// TIA Portal V15.1 export
// export: Created 2024-05-17T05:38:36.150876Z, ExportSetting WithDefaults, DisplayName Totally Integrated Automation Portal, DisplayVersion V15.1 Update 5, DisplayName TIA Portal Openness, DisplayVersion V15.1 Update 5, DisplayName SINAMICS Startdrive Advanced, DisplayVersion V15.1, DisplayName G130, G150, S120, S150, SINAMICS MV, S210, DisplayVersion V15.1, DisplayName G110M, G120, G120C, G120D, G120P, DisplayVersion V15.1, DisplayName STEP 7 Professional, DisplayVersion V15.1 Update 5, DisplayName STEP 7 Safety, DisplayVersion V15.1, DisplayName WinCC Professional, DisplayVersion V15.1 Update 5, DisplayName SIMATIC Visualization Architect, DisplayVersion V15.1
FUNCTION_BLOCK "LProcGeneralFunc"   // FB1738, FBD
TITLE = LProcGeneralFunc
{ S7_Optimized_Access := 'TRUE' }
AUTHOR : VCC
FAMILY : Control
NAME : Genfunc
VERSION : 0.1
// ================================================================================
// This module handles General Reverse Switch, General High Speed and Lamptest.
// It will also give the user and 8 bit interface for project specific functions.
// ================================================================================
// stored: AutoNumber false, IsIECCheckEnabled false, IsRetainMemResEnabled false, MemoryReserve 100, SetENOAutomatically False, UDAEnableTagReadback false
   VAR_INPUT
      I_GenRevSw { ExternalAccessible := 'False'; ExternalVisible := 'False'; ExternalWritable := 'False'} : Bool;   // General reverse switch
      I_GenHighSpeed { ExternalAccessible := 'False'; ExternalVisible := 'False'; ExternalWritable := 'False'} : Bool;   // General high speed
      I_Lamptest { ExternalAccessible := 'False'; ExternalVisible := 'False'; ExternalWritable := 'False'} : Bool;   // Lamptest PB
      I_ManualMode { ExternalAccessible := 'False'; ExternalVisible := 'False'; ExternalWritable := 'False'} : Bool := TRUE;   // Manual mode active
      I_LamptestSec { ExternalAccessible := 'False'; ExternalVisible := 'False'; ExternalWritable := 'False'} : Int := 60;   // The number of seconds that Lamptest will be on (Sec)
   END_VAR
   VAR_OUTPUT
      O_GeneralFunc : Word;   // General functions
      O_Lamptest { ExternalAccessible := 'False'; ExternalVisible := 'False'; ExternalWritable := 'False'} : Bool;   // Lamptest
      O_LamptestSteady { ExternalAccessible := 'False'; ExternalVisible := 'False'; ExternalWritable := 'False'} : Bool;   // Lamptest always on
      O_GenHighSpeed { ExternalAccessible := 'False'; ExternalVisible := 'False'; ExternalWritable := 'False'} : Bool;   // General High Speed
      O_GenRevSwitch { ExternalAccessible := 'False'; ExternalVisible := 'False'; ExternalWritable := 'False'} : Bool;   // Reverse Switch
      O_GenReverseAlarm { ExternalAccessible := 'False'; ExternalVisible := 'False'; ExternalWritable := 'False'} : Bool;   // Alarm when general reverse switch is ON while NOT in Manual mode
   END_VAR
   VAR DB_SPECIFIC
      H_HMIGenFuncCmd : Word;   // General function commands from HMI
      AutoMode { ExternalAccessible := 'False'; ExternalVisible := 'False'; ExternalWritable := 'False'} : Bool;   // Auto mode
      AutoSel { ExternalAccessible := 'False'; ExternalVisible := 'False'; ExternalWritable := 'False'} : Bool;   // Auto is selected
      AlarmAB { ExternalAccessible := 'False'; ExternalVisible := 'False'; ExternalWritable := 'False'} : Bool;   // Alarm A or B is active
      HMIGenHighSpeed { ExternalAccessible := 'False'; ExternalVisible := 'False'; ExternalWritable := 'False'} : Bool;   // General High Speed for manual movement
      HMILamptest { ExternalAccessible := 'False'; ExternalVisible := 'False'; ExternalWritable := 'False'} : Bool;   // Lamptest
      GenHighSpeedSelected { ExternalAccessible := 'False'; ExternalVisible := 'False'; ExternalWritable := 'False'} : Bool;   // General high speed is selected
      LamptestSelected : Bool;   // Lamptest is selected
      PulseLamptest { ExternalAccessible := 'False'; ExternalVisible := 'False'; ExternalWritable := 'False'} : Bool;   // Pulse for lamptest
      PulseGenHighSpeed { ExternalAccessible := 'False'; ExternalVisible := 'False'; ExternalWritable := 'False'} : Bool;   // Pulse General high speed
      TimerLamptest { ExternalAccessible := 'False'; ExternalVisible := 'False'; ExternalWritable := 'False'} : Bool;   // Timer for Lamptest
      LamptestSec { ExternalAccessible := 'False'; ExternalVisible := 'False'; ExternalWritable := 'False'} : DInt;   // Lamptest on for xxx milliesec
      LamptestMillieSec { ExternalAccessible := 'False'; ExternalVisible := 'False'; ExternalWritable := 'False'} : DInt;   // Converted value
   END_VAR
   VAR
      TimerLampTestSel { ExternalAccessible := 'False'; ExternalVisible := 'False'; ExternalWritable := 'False'; S7_SetPoint := 'True'} : "LTimer";
   END_VAR
   VAR_TEMP
      SetLamptest : Bool;   // Set Lamptest
      ResetLamptest : Bool;   // Reset Lamptest
      ElapseTime : DInt;   // Elapse time for Lamptest
   END_VAR
   VAR_TEMP   // added for the SCL form of the ladder/FBD networks
      _w1 : Bool;
      _w2 : Bool;
   END_VAR
BEGIN

REGION Network 1: **** 1 - Inputs **** Extract the general functions from HMI
   // Extract the general functions from HMI
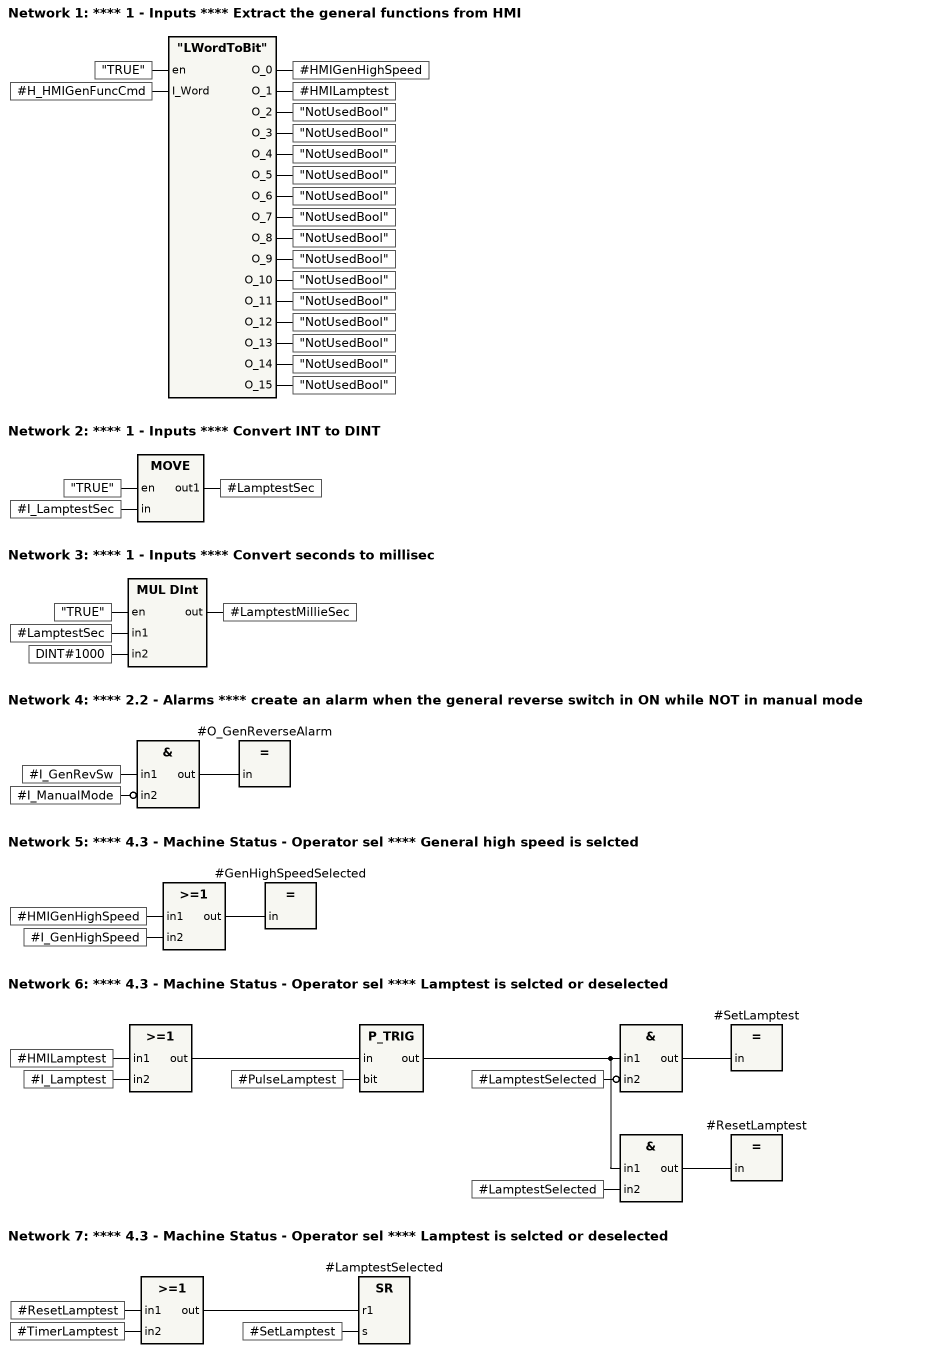
   IF "TRUE" THEN
       "LWordToBit"(I_Word := #H_HMIGenFuncCmd,
                    O_0 => #HMIGenHighSpeed,
                    O_1 => #HMILamptest,
                    O_2 => "NotUsedBool",
                    O_3 => "NotUsedBool",
                    O_4 => "NotUsedBool",
                    O_5 => "NotUsedBool",
                    O_6 => "NotUsedBool",
                    O_7 => "NotUsedBool",
                    O_8 => "NotUsedBool",
                    O_9 => "NotUsedBool",
                    O_10 => "NotUsedBool",
                    O_11 => "NotUsedBool",
                    O_12 => "NotUsedBool",
                    O_13 => "NotUsedBool",
                    O_14 => "NotUsedBool",
                    O_15 => "NotUsedBool");
   END_IF;
END_REGION

REGION Network 2: **** 1 - Inputs **** Convert INT to DINT
   // Convert INT to DINT
   IF "TRUE" THEN #LamptestSec := #I_LamptestSec; END_IF;
END_REGION

REGION Network 3: **** 1 - Inputs **** Convert seconds to millisec
   // Convert seconds to millisec
   IF "TRUE" THEN #LamptestMillieSec := #LamptestSec * DINT#1000; END_IF;
END_REGION

REGION Network 4: **** 2.2 - Alarms **** create an alarm when the general reverse switch in ON while NOT in manual mode
   // create an alarm when the general reverse switch in ON while NOT in manual mode
   #O_GenReverseAlarm := #I_GenRevSw AND NOT #I_ManualMode;
END_REGION

REGION Network 5: **** 4.3 - Machine Status - Operator sel **** General high speed is selcted
   // General high speed is selcted
   #GenHighSpeedSelected := #HMIGenHighSpeed OR #I_GenHighSpeed;
END_REGION

REGION Network 6: **** 4.3 - Machine Status - Operator sel **** Lamptest is selcted or deselected
   // Lamptest is selcted or deselected
   #_w1 := #HMILamptest OR #I_Lamptest;
   #_w2 := #_w1 AND NOT #PulseLamptest;   // rising edge
   #PulseLamptest := #_w1;
   #SetLamptest := #_w2 AND NOT #LamptestSelected;
   #ResetLamptest := #_w2 AND #LamptestSelected;
END_REGION

REGION Network 7: **** 4.3 - Machine Status - Operator sel **** Lamptest is selcted or deselected
   // Lamptest is selcted or deselected
   IF #SetLamptest THEN
       #LamptestSelected := TRUE;   // SR flip-flop
   END_IF;
   IF #ResetLamptest OR #TimerLamptest THEN #LamptestSelected := FALSE; END_IF;
END_REGION

REGION Network 8: **** 4.3 - Machine Status - Operator sel **** Timer for Lamptest
   // Timer for Lamptest
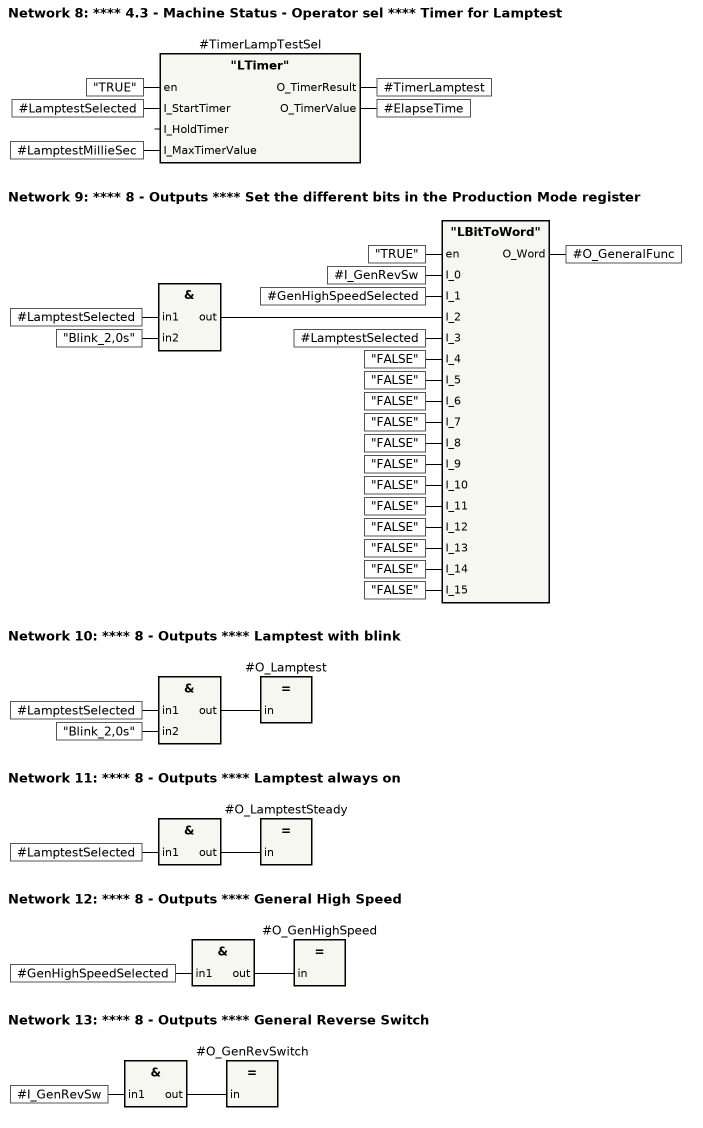
   IF "TRUE" THEN
       #TimerLampTestSel(I_StartTimer := #LamptestSelected,   // "LTimer"
                         I_MaxTimerValue := #LamptestMillieSec,
                         O_TimerResult => #TimerLamptest,
                         O_TimerValue => #ElapseTime);
   END_IF;
END_REGION

REGION Network 9: **** 8 - Outputs **** Set the different bits in the Production Mode register
   // Set the different bits in the Production Mode register
   IF "TRUE" THEN
       "LBitToWord"(I_0 := #I_GenRevSw,
                    I_1 := #GenHighSpeedSelected,
                    I_2 := #LamptestSelected AND "Blink_2,0s",
                    I_3 := #LamptestSelected,
                    I_4 := "FALSE",
                    I_5 := "FALSE",
                    I_6 := "FALSE",
                    I_7 := "FALSE",
                    I_8 := "FALSE",
                    I_9 := "FALSE",
                    I_10 := "FALSE",
                    I_11 := "FALSE",
                    I_12 := "FALSE",
                    I_13 := "FALSE",
                    I_14 := "FALSE",
                    I_15 := "FALSE",
                    O_Word => #O_GeneralFunc);
   END_IF;
END_REGION

REGION Network 10: **** 8 - Outputs **** Lamptest with blink
   // Lamptest with blink
   #O_Lamptest := #LamptestSelected AND "Blink_2,0s";
END_REGION

REGION Network 11: **** 8 - Outputs **** Lamptest always on
   // Lamptest always on
   #O_LamptestSteady := #LamptestSelected;
END_REGION

REGION Network 12: **** 8 - Outputs **** General High Speed
   // General High Speed
   #O_GenHighSpeed := #GenHighSpeedSelected;
END_REGION

REGION Network 13: **** 8 - Outputs **** General Reverse Switch
   // General Reverse Switch
   #O_GenRevSwitch := #I_GenRevSw;
END_REGION
END_FUNCTION_BLOCK
